FUNCTION ConsumeTime : bool
VAR_INPUT
	DelayUs 	: UDINT;
END_VAR
VAR
	fbGetTime	: GETCPUACCOUNT;
	tStart		: UDINT;
	tNow		: UDINT;
END_VAR

fbGetTime(cpuAccountDW => tStart);
tNow := tStart;

WHILE (tNow - tStart) < DelayUs*10 DO
	fbGetTime(cpuAccountDW => tNow);
END_WHILE

END_FUNCTION

(* stored: Version 1.1.0.1, ProductVersion 3.1.4024.11
   POU ConsumeTime: Id {efd0f232-f22a-4579-bec9-9dd5593716e8}, SpecialFunc None *)
